FUNCTION TANK_VOL1 : REAL
VAR_INPUT
	TR : REAL;
	TL : REAL;
	H : REAL;
END_VAR


(*
version 1.0	10. Mar 2010
programmer 	hugo
tested by		tobias

TANK_VOL1 calculates the volume of a tubular tank filled to level H.


*)

TANK_VOL1 := CIRCLE_SEG(TR, H) * TL;


(* revision histroy
hm	10. mar 2010	rev 1.0
	original version

*)

END_FUNCTION

(* stored: Version 1.1.0.1, ProductVersion 3.1.4022.7
   POU TANK_VOL1: Id {1c5b8dcd-c531-409d-8575-3949b6b78ae0}, SpecialFunc None *)
